(*

## Short summary

A basic datatype for physical parameters. It has just a value. 

.. <legal notes>

legal notes
=================
| SPDX-FileCopyrightText: © 2025 ekvip automation GmbH <info@ekvip.de>
| SPDX-License-Identifier: Apache-2.0
| For details check: Apache-2.0_

.. _Apache-2.0: https://www.apache.org/licenses/LICENSE-2.0

.. </legal notes>	

*)

TYPE BaseParameter :
STRUCT
	value :LREAL := 0.0;
END_STRUCT
END_TYPE

(* stored: Version 1.1.0.1
   DUT BaseParameter: Id {ac568200-85aa-4e07-b605-6de0a8afd9ad} *)
